// TIA Portal V19 export
FUNCTION "AUTO ALARM" : Void   // FC17, LAD
{ S7_Optimized_Access := 'TRUE' }
// stored: SetENOAutomatically false
BEGIN

REGION Network 1: ///////////////////////////////MFG PUPUP/////////////////////////////////////
END_REGION

REGION Network 2: PURIFIED WATER PROCESS SELECT
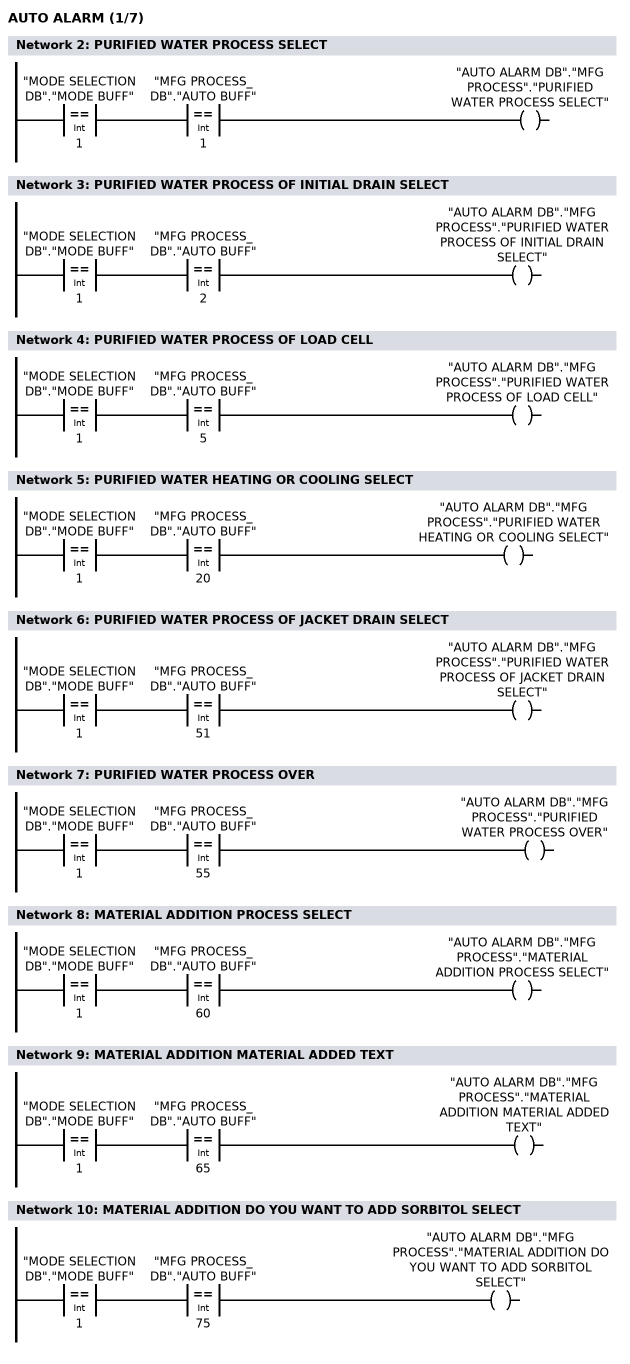
   RUNG wire#powerrail
      { S7_Templates := "SrcType := Int" } EQ_Contact(in1 := "MODE SELECTION DB"."MODE BUFF", in2 := 1)
      { S7_Templates := "SrcType := Int" } EQ_Contact(in1 := "MFG PROCESS_DB"."AUTO BUFF", in2 := 1)
      Coil( "AUTO ALARM DB"."MFG PROCESS"."PURIFIED WATER PROCESS SELECT" )
   END_RUNG
   // the same network as SCL:
   "AUTO ALARM DB"."MFG PROCESS"."PURIFIED WATER PROCESS SELECT" := ("MODE SELECTION DB"."MODE BUFF" = 1) AND ("MFG PROCESS_DB"."AUTO BUFF" = 1);
END_REGION

REGION Network 3: PURIFIED WATER PROCESS OF INITIAL DRAIN SELECT
   RUNG wire#powerrail
      { S7_Templates := "SrcType := Int" } EQ_Contact(in1 := "MODE SELECTION DB"."MODE BUFF", in2 := 1)
      { S7_Templates := "SrcType := Int" } EQ_Contact(in1 := "MFG PROCESS_DB"."AUTO BUFF", in2 := 2)
      Coil( "AUTO ALARM DB"."MFG PROCESS"."PURIFIED WATER PROCESS OF INITIAL DRAIN SELECT" )
   END_RUNG
   // the same network as SCL:
   "AUTO ALARM DB"."MFG PROCESS"."PURIFIED WATER PROCESS OF INITIAL DRAIN SELECT" := ("MODE SELECTION DB"."MODE BUFF" = 1) AND ("MFG PROCESS_DB"."AUTO BUFF" = 2);
END_REGION

REGION Network 4: PURIFIED WATER PROCESS OF LOAD CELL
   RUNG wire#powerrail
      { S7_Templates := "SrcType := Int" } EQ_Contact(in1 := "MODE SELECTION DB"."MODE BUFF", in2 := 1)
      { S7_Templates := "SrcType := Int" } EQ_Contact(in1 := "MFG PROCESS_DB"."AUTO BUFF", in2 := 5)
      Coil( "AUTO ALARM DB"."MFG PROCESS"."PURIFIED WATER PROCESS OF LOAD CELL" )
   END_RUNG
   // the same network as SCL:
   "AUTO ALARM DB"."MFG PROCESS"."PURIFIED WATER PROCESS OF LOAD CELL" := ("MODE SELECTION DB"."MODE BUFF" = 1) AND ("MFG PROCESS_DB"."AUTO BUFF" = 5);
END_REGION

REGION Network 5: PURIFIED WATER HEATING OR COOLING SELECT
   RUNG wire#powerrail
      { S7_Templates := "SrcType := Int" } EQ_Contact(in1 := "MODE SELECTION DB"."MODE BUFF", in2 := 1)
      { S7_Templates := "SrcType := Int" } EQ_Contact(in1 := "MFG PROCESS_DB"."AUTO BUFF", in2 := 20)
      Coil( "AUTO ALARM DB"."MFG PROCESS"."PURIFIED WATER HEATING OR COOLING SELECT" )
   END_RUNG
   // the same network as SCL:
   "AUTO ALARM DB"."MFG PROCESS"."PURIFIED WATER HEATING OR COOLING SELECT" := ("MODE SELECTION DB"."MODE BUFF" = 1) AND ("MFG PROCESS_DB"."AUTO BUFF" = 20);
END_REGION

REGION Network 6: PURIFIED WATER PROCESS OF JACKET DRAIN SELECT
   RUNG wire#powerrail
      { S7_Templates := "SrcType := Int" } EQ_Contact(in1 := "MODE SELECTION DB"."MODE BUFF", in2 := 1)
      { S7_Templates := "SrcType := Int" } EQ_Contact(in1 := "MFG PROCESS_DB"."AUTO BUFF", in2 := 51)
      Coil( "AUTO ALARM DB"."MFG PROCESS"."PURIFIED WATER PROCESS OF JACKET DRAIN SELECT" )
   END_RUNG
   // the same network as SCL:
   "AUTO ALARM DB"."MFG PROCESS"."PURIFIED WATER PROCESS OF JACKET DRAIN SELECT" := ("MODE SELECTION DB"."MODE BUFF" = 1) AND ("MFG PROCESS_DB"."AUTO BUFF" = 51);
END_REGION

REGION Network 7: PURIFIED WATER PROCESS OVER
   RUNG wire#powerrail
      { S7_Templates := "SrcType := Int" } EQ_Contact(in1 := "MODE SELECTION DB"."MODE BUFF", in2 := 1)
      { S7_Templates := "SrcType := Int" } EQ_Contact(in1 := "MFG PROCESS_DB"."AUTO BUFF", in2 := 55)
      Coil( "AUTO ALARM DB"."MFG PROCESS"."PURIFIED WATER PROCESS OVER" )
   END_RUNG
   // the same network as SCL:
   "AUTO ALARM DB"."MFG PROCESS"."PURIFIED WATER PROCESS OVER" := ("MODE SELECTION DB"."MODE BUFF" = 1) AND ("MFG PROCESS_DB"."AUTO BUFF" = 55);
END_REGION

REGION Network 8: MATERIAL ADDITION PROCESS SELECT
   RUNG wire#powerrail
      { S7_Templates := "SrcType := Int" } EQ_Contact(in1 := "MODE SELECTION DB"."MODE BUFF", in2 := 1)
      { S7_Templates := "SrcType := Int" } EQ_Contact(in1 := "MFG PROCESS_DB"."AUTO BUFF", in2 := 60)
      Coil( "AUTO ALARM DB"."MFG PROCESS"."MATERIAL ADDITION PROCESS SELECT" )
   END_RUNG
   // the same network as SCL:
   "AUTO ALARM DB"."MFG PROCESS"."MATERIAL ADDITION PROCESS SELECT" := ("MODE SELECTION DB"."MODE BUFF" = 1) AND ("MFG PROCESS_DB"."AUTO BUFF" = 60);
END_REGION

REGION Network 9: MATERIAL ADDITION MATERIAL ADDED TEXT
   RUNG wire#powerrail
      { S7_Templates := "SrcType := Int" } EQ_Contact(in1 := "MODE SELECTION DB"."MODE BUFF", in2 := 1)
      { S7_Templates := "SrcType := Int" } EQ_Contact(in1 := "MFG PROCESS_DB"."AUTO BUFF", in2 := 65)
      Coil( "AUTO ALARM DB"."MFG PROCESS"."MATERIAL ADDITION MATERIAL ADDED TEXT" )
   END_RUNG
   // the same network as SCL:
   "AUTO ALARM DB"."MFG PROCESS"."MATERIAL ADDITION MATERIAL ADDED TEXT" := ("MODE SELECTION DB"."MODE BUFF" = 1) AND ("MFG PROCESS_DB"."AUTO BUFF" = 65);
END_REGION

REGION Network 10: MATERIAL ADDITION DO YOU WANT TO ADD SORBITOL SELECT
   RUNG wire#powerrail
      { S7_Templates := "SrcType := Int" } EQ_Contact(in1 := "MODE SELECTION DB"."MODE BUFF", in2 := 1)
      { S7_Templates := "SrcType := Int" } EQ_Contact(in1 := "MFG PROCESS_DB"."AUTO BUFF", in2 := 75)
      Coil( "AUTO ALARM DB"."MFG PROCESS"."MATERIAL ADDITION DO YOU WANT TO ADD SORBITOL SELECT" )
   END_RUNG
   // the same network as SCL:
   "AUTO ALARM DB"."MFG PROCESS"."MATERIAL ADDITION DO YOU WANT TO ADD SORBITOL SELECT" := ("MODE SELECTION DB"."MODE BUFF" = 1) AND ("MFG PROCESS_DB"."AUTO BUFF" = 75);
END_REGION

REGION Network 11: MATERIAL ADDITION OF SORBITOL OVER
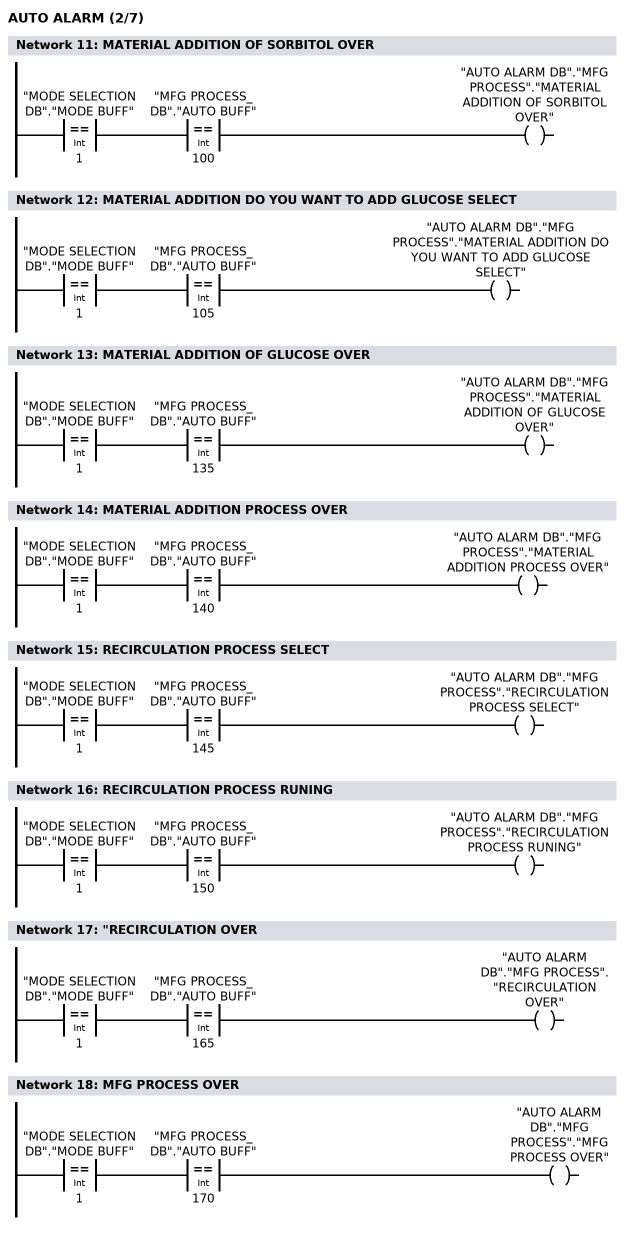
   RUNG wire#powerrail
      { S7_Templates := "SrcType := Int" } EQ_Contact(in1 := "MODE SELECTION DB"."MODE BUFF", in2 := 1)
      { S7_Templates := "SrcType := Int" } EQ_Contact(in1 := "MFG PROCESS_DB"."AUTO BUFF", in2 := 100)
      Coil( "AUTO ALARM DB"."MFG PROCESS"."MATERIAL ADDITION OF SORBITOL OVER" )
   END_RUNG
   // the same network as SCL:
   "AUTO ALARM DB"."MFG PROCESS"."MATERIAL ADDITION OF SORBITOL OVER" := ("MODE SELECTION DB"."MODE BUFF" = 1) AND ("MFG PROCESS_DB"."AUTO BUFF" = 100);
END_REGION

REGION Network 12: MATERIAL ADDITION DO YOU WANT TO ADD GLUCOSE SELECT
   RUNG wire#powerrail
      { S7_Templates := "SrcType := Int" } EQ_Contact(in1 := "MODE SELECTION DB"."MODE BUFF", in2 := 1)
      { S7_Templates := "SrcType := Int" } EQ_Contact(in1 := "MFG PROCESS_DB"."AUTO BUFF", in2 := 105)
      Coil( "AUTO ALARM DB"."MFG PROCESS"."MATERIAL ADDITION DO YOU WANT TO ADD GLUCOSE SELECT" )
   END_RUNG
   // the same network as SCL:
   "AUTO ALARM DB"."MFG PROCESS"."MATERIAL ADDITION DO YOU WANT TO ADD GLUCOSE SELECT" := ("MODE SELECTION DB"."MODE BUFF" = 1) AND ("MFG PROCESS_DB"."AUTO BUFF" = 105);
END_REGION

REGION Network 13: MATERIAL ADDITION OF GLUCOSE OVER
   RUNG wire#powerrail
      { S7_Templates := "SrcType := Int" } EQ_Contact(in1 := "MODE SELECTION DB"."MODE BUFF", in2 := 1)
      { S7_Templates := "SrcType := Int" } EQ_Contact(in1 := "MFG PROCESS_DB"."AUTO BUFF", in2 := 135)
      Coil( "AUTO ALARM DB"."MFG PROCESS"."MATERIAL ADDITION OF GLUCOSE OVER" )
   END_RUNG
   // the same network as SCL:
   "AUTO ALARM DB"."MFG PROCESS"."MATERIAL ADDITION OF GLUCOSE OVER" := ("MODE SELECTION DB"."MODE BUFF" = 1) AND ("MFG PROCESS_DB"."AUTO BUFF" = 135);
END_REGION

REGION Network 14: MATERIAL ADDITION PROCESS OVER
   RUNG wire#powerrail
      { S7_Templates := "SrcType := Int" } EQ_Contact(in1 := "MODE SELECTION DB"."MODE BUFF", in2 := 1)
      { S7_Templates := "SrcType := Int" } EQ_Contact(in1 := "MFG PROCESS_DB"."AUTO BUFF", in2 := 140)
      Coil( "AUTO ALARM DB"."MFG PROCESS"."MATERIAL ADDITION PROCESS OVER" )
   END_RUNG
   // the same network as SCL:
   "AUTO ALARM DB"."MFG PROCESS"."MATERIAL ADDITION PROCESS OVER" := ("MODE SELECTION DB"."MODE BUFF" = 1) AND ("MFG PROCESS_DB"."AUTO BUFF" = 140);
END_REGION

REGION Network 15: RECIRCULATION PROCESS SELECT
   RUNG wire#powerrail
      { S7_Templates := "SrcType := Int" } EQ_Contact(in1 := "MODE SELECTION DB"."MODE BUFF", in2 := 1)
      { S7_Templates := "SrcType := Int" } EQ_Contact(in1 := "MFG PROCESS_DB"."AUTO BUFF", in2 := 145)
      Coil( "AUTO ALARM DB"."MFG PROCESS"."RECIRCULATION PROCESS SELECT" )
   END_RUNG
   // the same network as SCL:
   "AUTO ALARM DB"."MFG PROCESS"."RECIRCULATION PROCESS SELECT" := ("MODE SELECTION DB"."MODE BUFF" = 1) AND ("MFG PROCESS_DB"."AUTO BUFF" = 145);
END_REGION

REGION Network 16: RECIRCULATION PROCESS RUNING
   RUNG wire#powerrail
      { S7_Templates := "SrcType := Int" } EQ_Contact(in1 := "MODE SELECTION DB"."MODE BUFF", in2 := 1)
      { S7_Templates := "SrcType := Int" } EQ_Contact(in1 := "MFG PROCESS_DB"."AUTO BUFF", in2 := 150)
      Coil( "AUTO ALARM DB"."MFG PROCESS"."RECIRCULATION PROCESS RUNING" )
   END_RUNG
   // the same network as SCL:
   "AUTO ALARM DB"."MFG PROCESS"."RECIRCULATION PROCESS RUNING" := ("MODE SELECTION DB"."MODE BUFF" = 1) AND ("MFG PROCESS_DB"."AUTO BUFF" = 150);
END_REGION

REGION Network 17: "RECIRCULATION OVER
   RUNG wire#powerrail
      { S7_Templates := "SrcType := Int" } EQ_Contact(in1 := "MODE SELECTION DB"."MODE BUFF", in2 := 1)
      { S7_Templates := "SrcType := Int" } EQ_Contact(in1 := "MFG PROCESS_DB"."AUTO BUFF", in2 := 165)
      Coil( "AUTO ALARM DB"."MFG PROCESS"."RECIRCULATION OVER" )
   END_RUNG
   // the same network as SCL:
   "AUTO ALARM DB"."MFG PROCESS"."RECIRCULATION OVER" := ("MODE SELECTION DB"."MODE BUFF" = 1) AND ("MFG PROCESS_DB"."AUTO BUFF" = 165);
END_REGION

REGION Network 18: MFG PROCESS OVER
   RUNG wire#powerrail
      { S7_Templates := "SrcType := Int" } EQ_Contact(in1 := "MODE SELECTION DB"."MODE BUFF", in2 := 1)
      { S7_Templates := "SrcType := Int" } EQ_Contact(in1 := "MFG PROCESS_DB"."AUTO BUFF", in2 := 170)
      Coil( "AUTO ALARM DB"."MFG PROCESS"."MFG PROCESS OVER" )
   END_RUNG
   // the same network as SCL:
   "AUTO ALARM DB"."MFG PROCESS"."MFG PROCESS OVER" := ("MODE SELECTION DB"."MODE BUFF" = 1) AND ("MFG PROCESS_DB"."AUTO BUFF" = 170);
END_REGION

REGION Network 20: TRANSFER START_MFG TO STORAGE ALL IN ONE FOR OVER (POPUP)
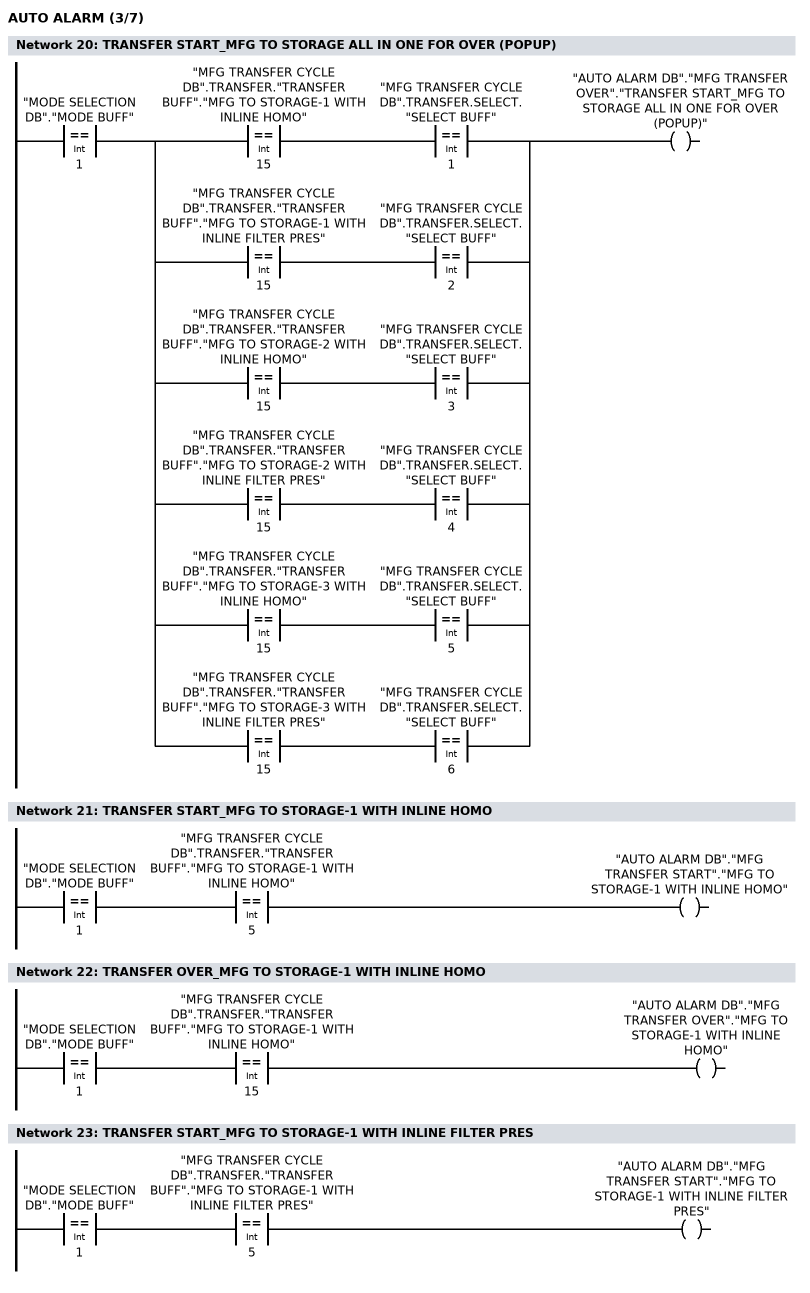
   RUNG wire#powerrail
      { S7_Templates := "SrcType := Int" } EQ_Contact(in1 := "MODE SELECTION DB"."MODE BUFF", in2 := 1)
      wire#w1
      { S7_Templates := "SrcType := Int" } EQ_Contact(in1 := "MFG TRANSFER CYCLE DB".TRANSFER."TRANSFER BUFF"."MFG TO STORAGE-1 WITH INLINE HOMO", in2 := 15)
      { S7_Templates := "SrcType := Int" } EQ_Contact(in1 := "MFG TRANSFER CYCLE DB".TRANSFER.SELECT."SELECT BUFF", in2 := 1)
      wire#w2
      Coil( "AUTO ALARM DB"."MFG TRANSFER OVER"."TRANSFER START_MFG TO STORAGE ALL IN ONE FOR OVER (POPUP)" )
   END_RUNG
   RUNG wire#w1
      { S7_Templates := "SrcType := Int" } EQ_Contact(in1 := "MFG TRANSFER CYCLE DB".TRANSFER."TRANSFER BUFF"."MFG TO STORAGE-1 WITH INLINE FILTER PRES", in2 := 15)
      { S7_Templates := "SrcType := Int" } EQ_Contact(in1 := "MFG TRANSFER CYCLE DB".TRANSFER.SELECT."SELECT BUFF", in2 := 2)
   END_RUNG wire#w2
   RUNG wire#w1
      { S7_Templates := "SrcType := Int" } EQ_Contact(in1 := "MFG TRANSFER CYCLE DB".TRANSFER."TRANSFER BUFF"."MFG TO STORAGE-2 WITH INLINE HOMO", in2 := 15)
      { S7_Templates := "SrcType := Int" } EQ_Contact(in1 := "MFG TRANSFER CYCLE DB".TRANSFER.SELECT."SELECT BUFF", in2 := 3)
   END_RUNG wire#w2
   RUNG wire#w1
      { S7_Templates := "SrcType := Int" } EQ_Contact(in1 := "MFG TRANSFER CYCLE DB".TRANSFER."TRANSFER BUFF"."MFG TO STORAGE-2 WITH INLINE FILTER PRES", in2 := 15)
      { S7_Templates := "SrcType := Int" } EQ_Contact(in1 := "MFG TRANSFER CYCLE DB".TRANSFER.SELECT."SELECT BUFF", in2 := 4)
   END_RUNG wire#w2
   RUNG wire#w1
      { S7_Templates := "SrcType := Int" } EQ_Contact(in1 := "MFG TRANSFER CYCLE DB".TRANSFER."TRANSFER BUFF"."MFG TO STORAGE-3 WITH INLINE HOMO", in2 := 15)
      { S7_Templates := "SrcType := Int" } EQ_Contact(in1 := "MFG TRANSFER CYCLE DB".TRANSFER.SELECT."SELECT BUFF", in2 := 5)
   END_RUNG wire#w2
   RUNG wire#w1
      { S7_Templates := "SrcType := Int" } EQ_Contact(in1 := "MFG TRANSFER CYCLE DB".TRANSFER."TRANSFER BUFF"."MFG TO STORAGE-3 WITH INLINE FILTER PRES", in2 := 15)
      { S7_Templates := "SrcType := Int" } EQ_Contact(in1 := "MFG TRANSFER CYCLE DB".TRANSFER.SELECT."SELECT BUFF", in2 := 6)
   END_RUNG wire#w2
   // the same network as SCL:
   "AUTO ALARM DB"."MFG TRANSFER OVER"."TRANSFER START_MFG TO STORAGE ALL IN ONE FOR OVER (POPUP)" := ("MODE SELECTION DB"."MODE BUFF" = 1) AND ((("MFG TRANSFER CYCLE DB".TRANSFER."TRANSFER BUFF"."MFG TO STORAGE-1 WITH INLINE HOMO" = 15) AND ("MFG TRANSFER CYCLE DB".TRANSFER.SELECT."SELECT BUFF" = 1)) OR (("MFG TRANSFER CYCLE DB".TRANSFER."TRANSFER BUFF"."MFG TO STORAGE-1 WITH INLINE FILTER PRES" = 15) AND ("MFG TRANSFER CYCLE DB".TRANSFER.SELECT."SELECT BUFF" = 2)) OR (("MFG TRANSFER CYCLE DB".TRANSFER."TRANSFER BUFF"."MFG TO STORAGE-2 WITH INLINE HOMO" = 15) AND ("MFG TRANSFER CYCLE DB".TRANSFER.SELECT."SELECT BUFF" = 3)) OR (("MFG TRANSFER CYCLE DB".TRANSFER."TRANSFER BUFF"."MFG TO STORAGE-2 WITH INLINE FILTER PRES" = 15) AND ("MFG TRANSFER CYCLE DB".TRANSFER.SELECT."SELECT BUFF" = 4)) OR (("MFG TRANSFER CYCLE DB".TRANSFER."TRANSFER BUFF"."MFG TO STORAGE-3 WITH INLINE HOMO" = 15) AND ("MFG TRANSFER CYCLE DB".TRANSFER.SELECT."SELECT BUFF" = 5)) OR (("MFG TRANSFER CYCLE DB".TRANSFER."TRANSFER BUFF"."MFG TO STORAGE-3 WITH INLINE FILTER PRES" = 15) AND ("MFG TRANSFER CYCLE DB".TRANSFER.SELECT."SELECT BUFF" = 6)));
END_REGION

REGION Network 21: TRANSFER START_MFG TO STORAGE-1 WITH INLINE HOMO
   RUNG wire#powerrail
      { S7_Templates := "SrcType := Int" } EQ_Contact(in1 := "MODE SELECTION DB"."MODE BUFF", in2 := 1)
      { S7_Templates := "SrcType := Int" } EQ_Contact(in1 := "MFG TRANSFER CYCLE DB".TRANSFER."TRANSFER BUFF"."MFG TO STORAGE-1 WITH INLINE HOMO", in2 := 5)
      Coil( "AUTO ALARM DB"."MFG TRANSFER START"."MFG TO STORAGE-1 WITH INLINE HOMO" )
   END_RUNG
   // the same network as SCL:
   "AUTO ALARM DB"."MFG TRANSFER START"."MFG TO STORAGE-1 WITH INLINE HOMO" := ("MODE SELECTION DB"."MODE BUFF" = 1) AND ("MFG TRANSFER CYCLE DB".TRANSFER."TRANSFER BUFF"."MFG TO STORAGE-1 WITH INLINE HOMO" = 5);
END_REGION

REGION Network 22: TRANSFER OVER_MFG TO STORAGE-1 WITH INLINE HOMO
   RUNG wire#powerrail
      { S7_Templates := "SrcType := Int" } EQ_Contact(in1 := "MODE SELECTION DB"."MODE BUFF", in2 := 1)
      { S7_Templates := "SrcType := Int" } EQ_Contact(in1 := "MFG TRANSFER CYCLE DB".TRANSFER."TRANSFER BUFF"."MFG TO STORAGE-1 WITH INLINE HOMO", in2 := 15)
      Coil( "AUTO ALARM DB"."MFG TRANSFER OVER"."MFG TO STORAGE-1 WITH INLINE HOMO" )
   END_RUNG
   // the same network as SCL:
   "AUTO ALARM DB"."MFG TRANSFER OVER"."MFG TO STORAGE-1 WITH INLINE HOMO" := ("MODE SELECTION DB"."MODE BUFF" = 1) AND ("MFG TRANSFER CYCLE DB".TRANSFER."TRANSFER BUFF"."MFG TO STORAGE-1 WITH INLINE HOMO" = 15);
END_REGION

REGION Network 23: TRANSFER START_MFG TO STORAGE-1 WITH INLINE FILTER PRES
   RUNG wire#powerrail
      { S7_Templates := "SrcType := Int" } EQ_Contact(in1 := "MODE SELECTION DB"."MODE BUFF", in2 := 1)
      { S7_Templates := "SrcType := Int" } EQ_Contact(in1 := "MFG TRANSFER CYCLE DB".TRANSFER."TRANSFER BUFF"."MFG TO STORAGE-1 WITH INLINE FILTER PRES", in2 := 5)
      Coil( "AUTO ALARM DB"."MFG TRANSFER START"."MFG TO STORAGE-1 WITH INLINE FILTER PRES" )
   END_RUNG
   // the same network as SCL:
   "AUTO ALARM DB"."MFG TRANSFER START"."MFG TO STORAGE-1 WITH INLINE FILTER PRES" := ("MODE SELECTION DB"."MODE BUFF" = 1) AND ("MFG TRANSFER CYCLE DB".TRANSFER."TRANSFER BUFF"."MFG TO STORAGE-1 WITH INLINE FILTER PRES" = 5);
END_REGION

REGION Network 24: TRANSFER OVER_MFG TO STORAGE-1 WITH INLINE FILTER PRES
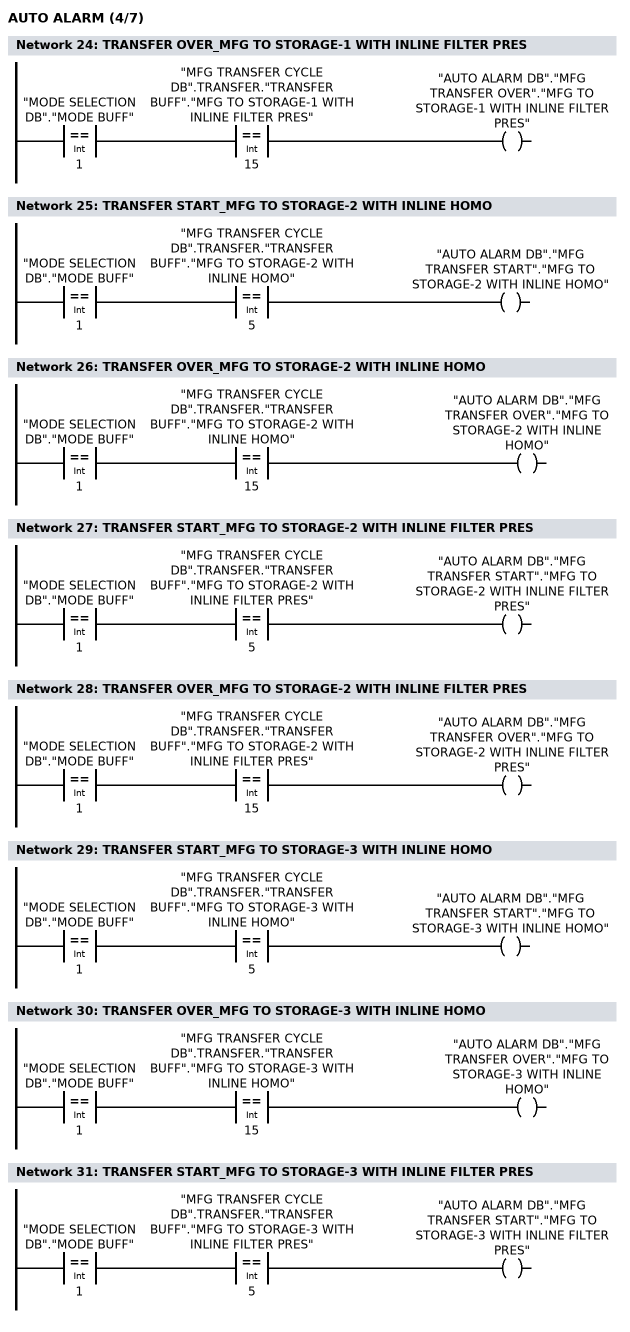
   RUNG wire#powerrail
      { S7_Templates := "SrcType := Int" } EQ_Contact(in1 := "MODE SELECTION DB"."MODE BUFF", in2 := 1)
      { S7_Templates := "SrcType := Int" } EQ_Contact(in1 := "MFG TRANSFER CYCLE DB".TRANSFER."TRANSFER BUFF"."MFG TO STORAGE-1 WITH INLINE FILTER PRES", in2 := 15)
      Coil( "AUTO ALARM DB"."MFG TRANSFER OVER"."MFG TO STORAGE-1 WITH INLINE FILTER PRES" )
   END_RUNG
   // the same network as SCL:
   "AUTO ALARM DB"."MFG TRANSFER OVER"."MFG TO STORAGE-1 WITH INLINE FILTER PRES" := ("MODE SELECTION DB"."MODE BUFF" = 1) AND ("MFG TRANSFER CYCLE DB".TRANSFER."TRANSFER BUFF"."MFG TO STORAGE-1 WITH INLINE FILTER PRES" = 15);
END_REGION

REGION Network 25: TRANSFER START_MFG TO STORAGE-2 WITH INLINE HOMO
   RUNG wire#powerrail
      { S7_Templates := "SrcType := Int" } EQ_Contact(in1 := "MODE SELECTION DB"."MODE BUFF", in2 := 1)
      { S7_Templates := "SrcType := Int" } EQ_Contact(in1 := "MFG TRANSFER CYCLE DB".TRANSFER."TRANSFER BUFF"."MFG TO STORAGE-2 WITH INLINE HOMO", in2 := 5)
      Coil( "AUTO ALARM DB"."MFG TRANSFER START"."MFG TO STORAGE-2 WITH INLINE HOMO" )
   END_RUNG
   // the same network as SCL:
   "AUTO ALARM DB"."MFG TRANSFER START"."MFG TO STORAGE-2 WITH INLINE HOMO" := ("MODE SELECTION DB"."MODE BUFF" = 1) AND ("MFG TRANSFER CYCLE DB".TRANSFER."TRANSFER BUFF"."MFG TO STORAGE-2 WITH INLINE HOMO" = 5);
END_REGION

REGION Network 26: TRANSFER OVER_MFG TO STORAGE-2 WITH INLINE HOMO
   RUNG wire#powerrail
      { S7_Templates := "SrcType := Int" } EQ_Contact(in1 := "MODE SELECTION DB"."MODE BUFF", in2 := 1)
      { S7_Templates := "SrcType := Int" } EQ_Contact(in1 := "MFG TRANSFER CYCLE DB".TRANSFER."TRANSFER BUFF"."MFG TO STORAGE-2 WITH INLINE HOMO", in2 := 15)
      Coil( "AUTO ALARM DB"."MFG TRANSFER OVER"."MFG TO STORAGE-2 WITH INLINE HOMO" )
   END_RUNG
   // the same network as SCL:
   "AUTO ALARM DB"."MFG TRANSFER OVER"."MFG TO STORAGE-2 WITH INLINE HOMO" := ("MODE SELECTION DB"."MODE BUFF" = 1) AND ("MFG TRANSFER CYCLE DB".TRANSFER."TRANSFER BUFF"."MFG TO STORAGE-2 WITH INLINE HOMO" = 15);
END_REGION

REGION Network 27: TRANSFER START_MFG TO STORAGE-2 WITH INLINE FILTER PRES
   RUNG wire#powerrail
      { S7_Templates := "SrcType := Int" } EQ_Contact(in1 := "MODE SELECTION DB"."MODE BUFF", in2 := 1)
      { S7_Templates := "SrcType := Int" } EQ_Contact(in1 := "MFG TRANSFER CYCLE DB".TRANSFER."TRANSFER BUFF"."MFG TO STORAGE-2 WITH INLINE FILTER PRES", in2 := 5)
      Coil( "AUTO ALARM DB"."MFG TRANSFER START"."MFG TO STORAGE-2 WITH INLINE FILTER PRES" )
   END_RUNG
   // the same network as SCL:
   "AUTO ALARM DB"."MFG TRANSFER START"."MFG TO STORAGE-2 WITH INLINE FILTER PRES" := ("MODE SELECTION DB"."MODE BUFF" = 1) AND ("MFG TRANSFER CYCLE DB".TRANSFER."TRANSFER BUFF"."MFG TO STORAGE-2 WITH INLINE FILTER PRES" = 5);
END_REGION

REGION Network 28: TRANSFER OVER_MFG TO STORAGE-2 WITH INLINE FILTER PRES
   RUNG wire#powerrail
      { S7_Templates := "SrcType := Int" } EQ_Contact(in1 := "MODE SELECTION DB"."MODE BUFF", in2 := 1)
      { S7_Templates := "SrcType := Int" } EQ_Contact(in1 := "MFG TRANSFER CYCLE DB".TRANSFER."TRANSFER BUFF"."MFG TO STORAGE-2 WITH INLINE FILTER PRES", in2 := 15)
      Coil( "AUTO ALARM DB"."MFG TRANSFER OVER"."MFG TO STORAGE-2 WITH INLINE FILTER PRES" )
   END_RUNG
   // the same network as SCL:
   "AUTO ALARM DB"."MFG TRANSFER OVER"."MFG TO STORAGE-2 WITH INLINE FILTER PRES" := ("MODE SELECTION DB"."MODE BUFF" = 1) AND ("MFG TRANSFER CYCLE DB".TRANSFER."TRANSFER BUFF"."MFG TO STORAGE-2 WITH INLINE FILTER PRES" = 15);
END_REGION

REGION Network 29: TRANSFER START_MFG TO STORAGE-3 WITH INLINE HOMO
   RUNG wire#powerrail
      { S7_Templates := "SrcType := Int" } EQ_Contact(in1 := "MODE SELECTION DB"."MODE BUFF", in2 := 1)
      { S7_Templates := "SrcType := Int" } EQ_Contact(in1 := "MFG TRANSFER CYCLE DB".TRANSFER."TRANSFER BUFF"."MFG TO STORAGE-3 WITH INLINE HOMO", in2 := 5)
      Coil( "AUTO ALARM DB"."MFG TRANSFER START"."MFG TO STORAGE-3 WITH INLINE HOMO" )
   END_RUNG
   // the same network as SCL:
   "AUTO ALARM DB"."MFG TRANSFER START"."MFG TO STORAGE-3 WITH INLINE HOMO" := ("MODE SELECTION DB"."MODE BUFF" = 1) AND ("MFG TRANSFER CYCLE DB".TRANSFER."TRANSFER BUFF"."MFG TO STORAGE-3 WITH INLINE HOMO" = 5);
END_REGION

REGION Network 30: TRANSFER OVER_MFG TO STORAGE-3 WITH INLINE HOMO
   RUNG wire#powerrail
      { S7_Templates := "SrcType := Int" } EQ_Contact(in1 := "MODE SELECTION DB"."MODE BUFF", in2 := 1)
      { S7_Templates := "SrcType := Int" } EQ_Contact(in1 := "MFG TRANSFER CYCLE DB".TRANSFER."TRANSFER BUFF"."MFG TO STORAGE-3 WITH INLINE HOMO", in2 := 15)
      Coil( "AUTO ALARM DB"."MFG TRANSFER OVER"."MFG TO STORAGE-3 WITH INLINE HOMO" )
   END_RUNG
   // the same network as SCL:
   "AUTO ALARM DB"."MFG TRANSFER OVER"."MFG TO STORAGE-3 WITH INLINE HOMO" := ("MODE SELECTION DB"."MODE BUFF" = 1) AND ("MFG TRANSFER CYCLE DB".TRANSFER."TRANSFER BUFF"."MFG TO STORAGE-3 WITH INLINE HOMO" = 15);
END_REGION

REGION Network 31: TRANSFER START_MFG TO STORAGE-3 WITH INLINE FILTER PRES
   RUNG wire#powerrail
      { S7_Templates := "SrcType := Int" } EQ_Contact(in1 := "MODE SELECTION DB"."MODE BUFF", in2 := 1)
      { S7_Templates := "SrcType := Int" } EQ_Contact(in1 := "MFG TRANSFER CYCLE DB".TRANSFER."TRANSFER BUFF"."MFG TO STORAGE-3 WITH INLINE FILTER PRES", in2 := 5)
      Coil( "AUTO ALARM DB"."MFG TRANSFER START"."MFG TO STORAGE-3 WITH INLINE FILTER PRES" )
   END_RUNG
   // the same network as SCL:
   "AUTO ALARM DB"."MFG TRANSFER START"."MFG TO STORAGE-3 WITH INLINE FILTER PRES" := ("MODE SELECTION DB"."MODE BUFF" = 1) AND ("MFG TRANSFER CYCLE DB".TRANSFER."TRANSFER BUFF"."MFG TO STORAGE-3 WITH INLINE FILTER PRES" = 5);
END_REGION

REGION Network 32: TRANSFER OVER_MFG TO STORAGE-3 WITH INLINE FILTER PRES
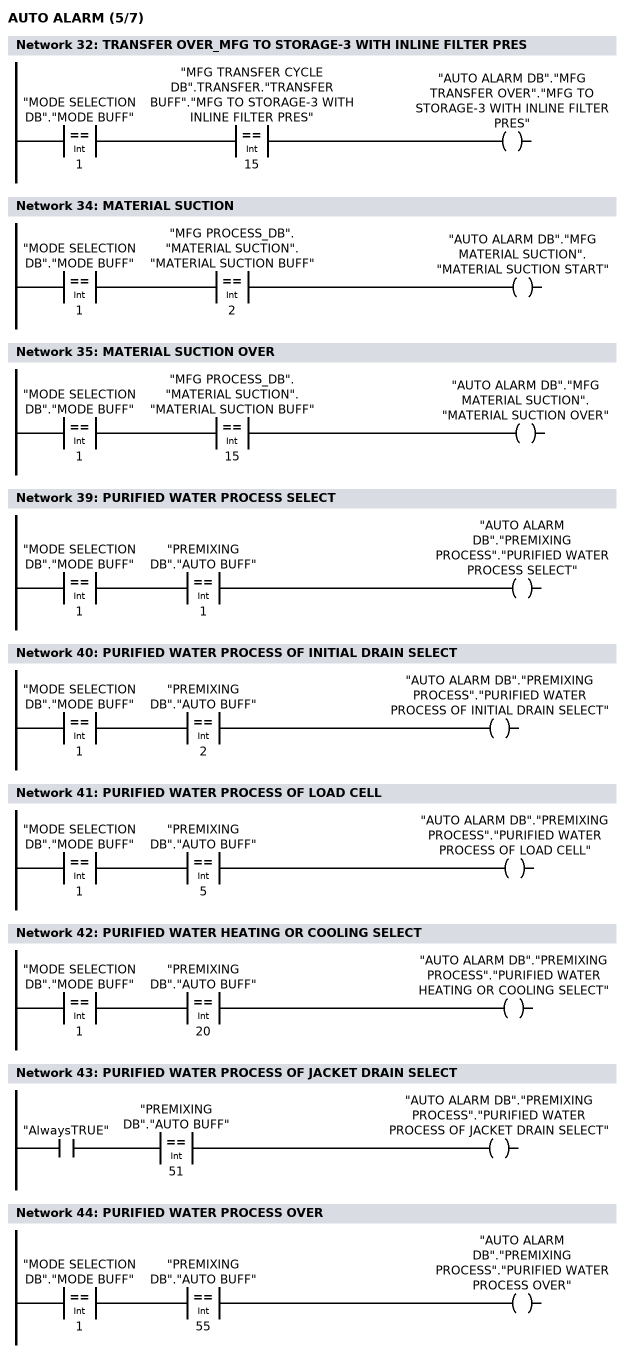
   RUNG wire#powerrail
      { S7_Templates := "SrcType := Int" } EQ_Contact(in1 := "MODE SELECTION DB"."MODE BUFF", in2 := 1)
      { S7_Templates := "SrcType := Int" } EQ_Contact(in1 := "MFG TRANSFER CYCLE DB".TRANSFER."TRANSFER BUFF"."MFG TO STORAGE-3 WITH INLINE FILTER PRES", in2 := 15)
      Coil( "AUTO ALARM DB"."MFG TRANSFER OVER"."MFG TO STORAGE-3 WITH INLINE FILTER PRES" )
   END_RUNG
   // the same network as SCL:
   "AUTO ALARM DB"."MFG TRANSFER OVER"."MFG TO STORAGE-3 WITH INLINE FILTER PRES" := ("MODE SELECTION DB"."MODE BUFF" = 1) AND ("MFG TRANSFER CYCLE DB".TRANSFER."TRANSFER BUFF"."MFG TO STORAGE-3 WITH INLINE FILTER PRES" = 15);
END_REGION

REGION Network 34: MATERIAL SUCTION
   RUNG wire#powerrail
      { S7_Templates := "SrcType := Int" } EQ_Contact(in1 := "MODE SELECTION DB"."MODE BUFF", in2 := 1)
      { S7_Templates := "SrcType := Int" } EQ_Contact(in1 := "MFG PROCESS_DB"."MATERIAL SUCTION"."MATERIAL SUCTION BUFF", in2 := 2)
      Coil( "AUTO ALARM DB"."MFG MATERIAL SUCTION"."MATERIAL SUCTION START" )
   END_RUNG
   // the same network as SCL:
   "AUTO ALARM DB"."MFG MATERIAL SUCTION"."MATERIAL SUCTION START" := ("MODE SELECTION DB"."MODE BUFF" = 1) AND ("MFG PROCESS_DB"."MATERIAL SUCTION"."MATERIAL SUCTION BUFF" = 2);
END_REGION

REGION Network 35: MATERIAL SUCTION OVER
   RUNG wire#powerrail
      { S7_Templates := "SrcType := Int" } EQ_Contact(in1 := "MODE SELECTION DB"."MODE BUFF", in2 := 1)
      { S7_Templates := "SrcType := Int" } EQ_Contact(in1 := "MFG PROCESS_DB"."MATERIAL SUCTION"."MATERIAL SUCTION BUFF", in2 := 15)
      Coil( "AUTO ALARM DB"."MFG MATERIAL SUCTION"."MATERIAL SUCTION OVER" )
   END_RUNG
   // the same network as SCL:
   "AUTO ALARM DB"."MFG MATERIAL SUCTION"."MATERIAL SUCTION OVER" := ("MODE SELECTION DB"."MODE BUFF" = 1) AND ("MFG PROCESS_DB"."MATERIAL SUCTION"."MATERIAL SUCTION BUFF" = 15);
END_REGION

REGION Network 38: /////////////////////////////// PREMIXING PUPUP /////////////////////////////////////
END_REGION

REGION Network 39: PURIFIED WATER PROCESS SELECT
   RUNG wire#powerrail
      { S7_Templates := "SrcType := Int" } EQ_Contact(in1 := "MODE SELECTION DB"."MODE BUFF", in2 := 1)
      { S7_Templates := "SrcType := Int" } EQ_Contact(in1 := "PREMIXING DB"."AUTO BUFF", in2 := 1)
      Coil( "AUTO ALARM DB"."PREMIXING PROCESS"."PURIFIED WATER PROCESS SELECT" )
   END_RUNG
   // the same network as SCL:
   "AUTO ALARM DB"."PREMIXING PROCESS"."PURIFIED WATER PROCESS SELECT" := ("MODE SELECTION DB"."MODE BUFF" = 1) AND ("PREMIXING DB"."AUTO BUFF" = 1);
END_REGION

REGION Network 40: PURIFIED WATER PROCESS OF INITIAL DRAIN SELECT
   RUNG wire#powerrail
      { S7_Templates := "SrcType := Int" } EQ_Contact(in1 := "MODE SELECTION DB"."MODE BUFF", in2 := 1)
      { S7_Templates := "SrcType := Int" } EQ_Contact(in1 := "PREMIXING DB"."AUTO BUFF", in2 := 2)
      Coil( "AUTO ALARM DB"."PREMIXING PROCESS"."PURIFIED WATER PROCESS OF INITIAL DRAIN SELECT" )
   END_RUNG
   // the same network as SCL:
   "AUTO ALARM DB"."PREMIXING PROCESS"."PURIFIED WATER PROCESS OF INITIAL DRAIN SELECT" := ("MODE SELECTION DB"."MODE BUFF" = 1) AND ("PREMIXING DB"."AUTO BUFF" = 2);
END_REGION

REGION Network 41: PURIFIED WATER PROCESS OF LOAD CELL
   RUNG wire#powerrail
      { S7_Templates := "SrcType := Int" } EQ_Contact(in1 := "MODE SELECTION DB"."MODE BUFF", in2 := 1)
      { S7_Templates := "SrcType := Int" } EQ_Contact(in1 := "PREMIXING DB"."AUTO BUFF", in2 := 5)
      Coil( "AUTO ALARM DB"."PREMIXING PROCESS"."PURIFIED WATER PROCESS OF LOAD CELL" )
   END_RUNG
   // the same network as SCL:
   "AUTO ALARM DB"."PREMIXING PROCESS"."PURIFIED WATER PROCESS OF LOAD CELL" := ("MODE SELECTION DB"."MODE BUFF" = 1) AND ("PREMIXING DB"."AUTO BUFF" = 5);
END_REGION

REGION Network 42: PURIFIED WATER HEATING OR COOLING SELECT
   RUNG wire#powerrail
      { S7_Templates := "SrcType := Int" } EQ_Contact(in1 := "MODE SELECTION DB"."MODE BUFF", in2 := 1)
      { S7_Templates := "SrcType := Int" } EQ_Contact(in1 := "PREMIXING DB"."AUTO BUFF", in2 := 20)
      Coil( "AUTO ALARM DB"."PREMIXING PROCESS"."PURIFIED WATER HEATING OR COOLING SELECT" )
   END_RUNG
   // the same network as SCL:
   "AUTO ALARM DB"."PREMIXING PROCESS"."PURIFIED WATER HEATING OR COOLING SELECT" := ("MODE SELECTION DB"."MODE BUFF" = 1) AND ("PREMIXING DB"."AUTO BUFF" = 20);
END_REGION

REGION Network 43: PURIFIED WATER PROCESS OF JACKET DRAIN SELECT
   RUNG wire#powerrail
      Contact( "AlwaysTRUE" )
      { S7_Templates := "SrcType := Int" } EQ_Contact(in1 := "PREMIXING DB"."AUTO BUFF", in2 := 51)
      Coil( "AUTO ALARM DB"."PREMIXING PROCESS"."PURIFIED WATER PROCESS OF JACKET DRAIN SELECT" )
   END_RUNG
   // the same network as SCL:
   "AUTO ALARM DB"."PREMIXING PROCESS"."PURIFIED WATER PROCESS OF JACKET DRAIN SELECT" := "AlwaysTRUE" AND ("PREMIXING DB"."AUTO BUFF" = 51);
END_REGION

REGION Network 44: PURIFIED WATER PROCESS OVER
   RUNG wire#powerrail
      { S7_Templates := "SrcType := Int" } EQ_Contact(in1 := "MODE SELECTION DB"."MODE BUFF", in2 := 1)
      { S7_Templates := "SrcType := Int" } EQ_Contact(in1 := "PREMIXING DB"."AUTO BUFF", in2 := 55)
      Coil( "AUTO ALARM DB"."PREMIXING PROCESS"."PURIFIED WATER PROCESS OVER" )
   END_RUNG
   // the same network as SCL:
   "AUTO ALARM DB"."PREMIXING PROCESS"."PURIFIED WATER PROCESS OVER" := ("MODE SELECTION DB"."MODE BUFF" = 1) AND ("PREMIXING DB"."AUTO BUFF" = 55);
END_REGION

REGION Network 45: MATERIAL ADDITION PROCESS SELECT
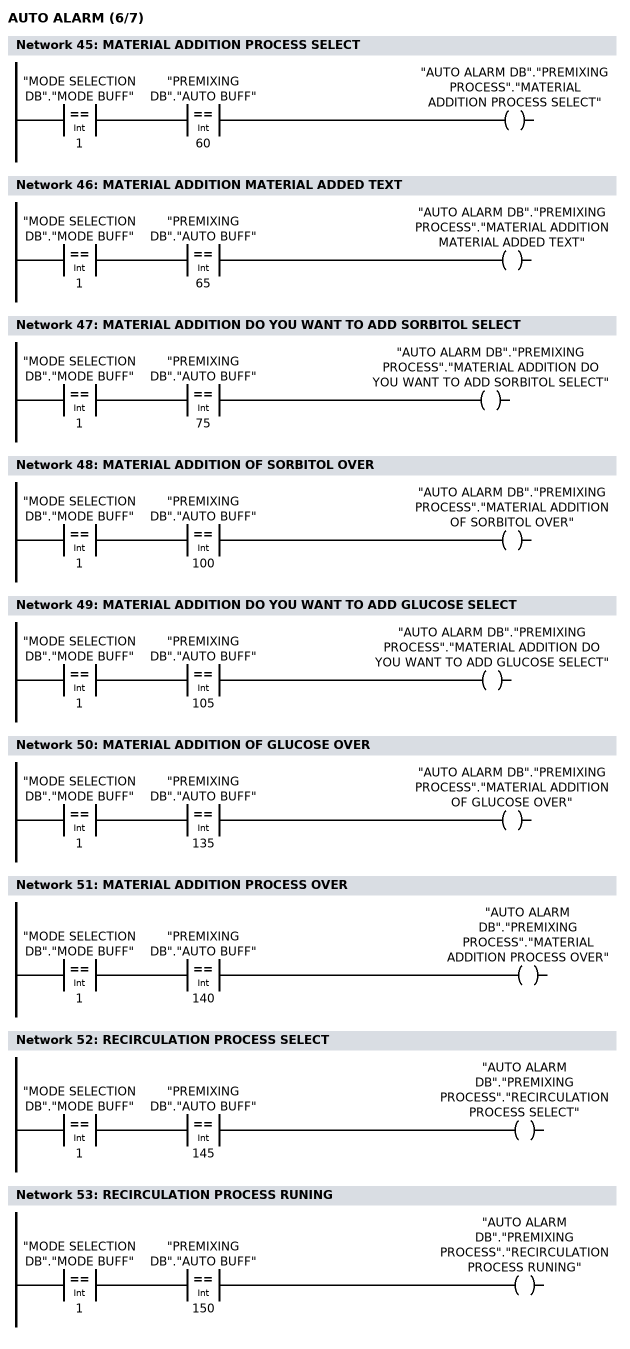
   RUNG wire#powerrail
      { S7_Templates := "SrcType := Int" } EQ_Contact(in1 := "MODE SELECTION DB"."MODE BUFF", in2 := 1)
      { S7_Templates := "SrcType := Int" } EQ_Contact(in1 := "PREMIXING DB"."AUTO BUFF", in2 := 60)
      Coil( "AUTO ALARM DB"."PREMIXING PROCESS"."MATERIAL ADDITION PROCESS SELECT" )
   END_RUNG
   // the same network as SCL:
   "AUTO ALARM DB"."PREMIXING PROCESS"."MATERIAL ADDITION PROCESS SELECT" := ("MODE SELECTION DB"."MODE BUFF" = 1) AND ("PREMIXING DB"."AUTO BUFF" = 60);
END_REGION

REGION Network 46: MATERIAL ADDITION MATERIAL ADDED TEXT
   RUNG wire#powerrail
      { S7_Templates := "SrcType := Int" } EQ_Contact(in1 := "MODE SELECTION DB"."MODE BUFF", in2 := 1)
      { S7_Templates := "SrcType := Int" } EQ_Contact(in1 := "PREMIXING DB"."AUTO BUFF", in2 := 65)
      Coil( "AUTO ALARM DB"."PREMIXING PROCESS"."MATERIAL ADDITION MATERIAL ADDED TEXT" )
   END_RUNG
   // the same network as SCL:
   "AUTO ALARM DB"."PREMIXING PROCESS"."MATERIAL ADDITION MATERIAL ADDED TEXT" := ("MODE SELECTION DB"."MODE BUFF" = 1) AND ("PREMIXING DB"."AUTO BUFF" = 65);
END_REGION

REGION Network 47: MATERIAL ADDITION DO YOU WANT TO ADD SORBITOL SELECT
   RUNG wire#powerrail
      { S7_Templates := "SrcType := Int" } EQ_Contact(in1 := "MODE SELECTION DB"."MODE BUFF", in2 := 1)
      { S7_Templates := "SrcType := Int" } EQ_Contact(in1 := "PREMIXING DB"."AUTO BUFF", in2 := 75)
      Coil( "AUTO ALARM DB"."PREMIXING PROCESS"."MATERIAL ADDITION DO YOU WANT TO ADD SORBITOL SELECT" )
   END_RUNG
   // the same network as SCL:
   "AUTO ALARM DB"."PREMIXING PROCESS"."MATERIAL ADDITION DO YOU WANT TO ADD SORBITOL SELECT" := ("MODE SELECTION DB"."MODE BUFF" = 1) AND ("PREMIXING DB"."AUTO BUFF" = 75);
END_REGION

REGION Network 48: MATERIAL ADDITION OF SORBITOL OVER
   RUNG wire#powerrail
      { S7_Templates := "SrcType := Int" } EQ_Contact(in1 := "MODE SELECTION DB"."MODE BUFF", in2 := 1)
      { S7_Templates := "SrcType := Int" } EQ_Contact(in1 := "PREMIXING DB"."AUTO BUFF", in2 := 100)
      Coil( "AUTO ALARM DB"."PREMIXING PROCESS"."MATERIAL ADDITION OF SORBITOL OVER" )
   END_RUNG
   // the same network as SCL:
   "AUTO ALARM DB"."PREMIXING PROCESS"."MATERIAL ADDITION OF SORBITOL OVER" := ("MODE SELECTION DB"."MODE BUFF" = 1) AND ("PREMIXING DB"."AUTO BUFF" = 100);
END_REGION

REGION Network 49: MATERIAL ADDITION DO YOU WANT TO ADD GLUCOSE SELECT
   RUNG wire#powerrail
      { S7_Templates := "SrcType := Int" } EQ_Contact(in1 := "MODE SELECTION DB"."MODE BUFF", in2 := 1)
      { S7_Templates := "SrcType := Int" } EQ_Contact(in1 := "PREMIXING DB"."AUTO BUFF", in2 := 105)
      Coil( "AUTO ALARM DB"."PREMIXING PROCESS"."MATERIAL ADDITION DO YOU WANT TO ADD GLUCOSE SELECT" )
   END_RUNG
   // the same network as SCL:
   "AUTO ALARM DB"."PREMIXING PROCESS"."MATERIAL ADDITION DO YOU WANT TO ADD GLUCOSE SELECT" := ("MODE SELECTION DB"."MODE BUFF" = 1) AND ("PREMIXING DB"."AUTO BUFF" = 105);
END_REGION

REGION Network 50: MATERIAL ADDITION OF GLUCOSE OVER
   RUNG wire#powerrail
      { S7_Templates := "SrcType := Int" } EQ_Contact(in1 := "MODE SELECTION DB"."MODE BUFF", in2 := 1)
      { S7_Templates := "SrcType := Int" } EQ_Contact(in1 := "PREMIXING DB"."AUTO BUFF", in2 := 135)
      Coil( "AUTO ALARM DB"."PREMIXING PROCESS"."MATERIAL ADDITION OF GLUCOSE OVER" )
   END_RUNG
   // the same network as SCL:
   "AUTO ALARM DB"."PREMIXING PROCESS"."MATERIAL ADDITION OF GLUCOSE OVER" := ("MODE SELECTION DB"."MODE BUFF" = 1) AND ("PREMIXING DB"."AUTO BUFF" = 135);
END_REGION

REGION Network 51: MATERIAL ADDITION PROCESS OVER
   RUNG wire#powerrail
      { S7_Templates := "SrcType := Int" } EQ_Contact(in1 := "MODE SELECTION DB"."MODE BUFF", in2 := 1)
      { S7_Templates := "SrcType := Int" } EQ_Contact(in1 := "PREMIXING DB"."AUTO BUFF", in2 := 140)
      Coil( "AUTO ALARM DB"."PREMIXING PROCESS"."MATERIAL ADDITION PROCESS OVER" )
   END_RUNG
   // the same network as SCL:
   "AUTO ALARM DB"."PREMIXING PROCESS"."MATERIAL ADDITION PROCESS OVER" := ("MODE SELECTION DB"."MODE BUFF" = 1) AND ("PREMIXING DB"."AUTO BUFF" = 140);
END_REGION

REGION Network 52: RECIRCULATION PROCESS SELECT
   RUNG wire#powerrail
      { S7_Templates := "SrcType := Int" } EQ_Contact(in1 := "MODE SELECTION DB"."MODE BUFF", in2 := 1)
      { S7_Templates := "SrcType := Int" } EQ_Contact(in1 := "PREMIXING DB"."AUTO BUFF", in2 := 145)
      Coil( "AUTO ALARM DB"."PREMIXING PROCESS"."RECIRCULATION PROCESS SELECT" )
   END_RUNG
   // the same network as SCL:
   "AUTO ALARM DB"."PREMIXING PROCESS"."RECIRCULATION PROCESS SELECT" := ("MODE SELECTION DB"."MODE BUFF" = 1) AND ("PREMIXING DB"."AUTO BUFF" = 145);
END_REGION

REGION Network 53: RECIRCULATION PROCESS RUNING
   RUNG wire#powerrail
      { S7_Templates := "SrcType := Int" } EQ_Contact(in1 := "MODE SELECTION DB"."MODE BUFF", in2 := 1)
      { S7_Templates := "SrcType := Int" } EQ_Contact(in1 := "PREMIXING DB"."AUTO BUFF", in2 := 150)
      Coil( "AUTO ALARM DB"."PREMIXING PROCESS"."RECIRCULATION PROCESS RUNING" )
   END_RUNG
   // the same network as SCL:
   "AUTO ALARM DB"."PREMIXING PROCESS"."RECIRCULATION PROCESS RUNING" := ("MODE SELECTION DB"."MODE BUFF" = 1) AND ("PREMIXING DB"."AUTO BUFF" = 150);
END_REGION

REGION Network 54: "RECIRCULATION OVER
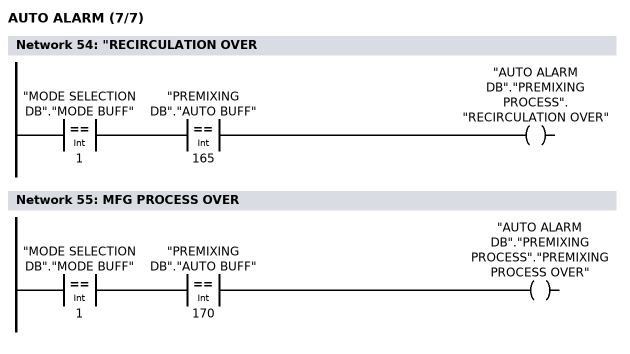
   RUNG wire#powerrail
      { S7_Templates := "SrcType := Int" } EQ_Contact(in1 := "MODE SELECTION DB"."MODE BUFF", in2 := 1)
      { S7_Templates := "SrcType := Int" } EQ_Contact(in1 := "PREMIXING DB"."AUTO BUFF", in2 := 165)
      Coil( "AUTO ALARM DB"."PREMIXING PROCESS"."RECIRCULATION OVER" )
   END_RUNG
   // the same network as SCL:
   "AUTO ALARM DB"."PREMIXING PROCESS"."RECIRCULATION OVER" := ("MODE SELECTION DB"."MODE BUFF" = 1) AND ("PREMIXING DB"."AUTO BUFF" = 165);
END_REGION

REGION Network 55: MFG PROCESS OVER
   RUNG wire#powerrail
      { S7_Templates := "SrcType := Int" } EQ_Contact(in1 := "MODE SELECTION DB"."MODE BUFF", in2 := 1)
      { S7_Templates := "SrcType := Int" } EQ_Contact(in1 := "PREMIXING DB"."AUTO BUFF", in2 := 170)
      Coil( "AUTO ALARM DB"."PREMIXING PROCESS"."PREMIXING PROCESS OVER" )
   END_RUNG
   // the same network as SCL:
   "AUTO ALARM DB"."PREMIXING PROCESS"."PREMIXING PROCESS OVER" := ("MODE SELECTION DB"."MODE BUFF" = 1) AND ("PREMIXING DB"."AUTO BUFF" = 170);
END_REGION
END_FUNCTION
